// TIA Portal V20 export
FUNCTION "LER_PartData_QrReaderPos" : Void   // FC10000, LAD
// stored: Access Published, SetENOAutomatically false
   VAR_INPUT
      generateCondition : Bool;
      PartOn : Bool;
      JudgmentOK : Bool;
      JudgmentNG : Bool;
      JudgmentBusy : Bool;
      QrReadData : String;
   END_VAR
   VAR_OUTPUT
      PartData : "LER_typePartData";
      ResultData : "LER_typeQrData";
   END_VAR
   VAR_TEMP
      tempRET_VAL : Word;
   END_VAR
   VAR CONSTANT
      PartStatus_Busy : Byte := 16#2;
      PartStatus_Ok : Byte := 16#3;
      PartStatus_NG : Byte := 16#4;
      TRUE : Bool := TRUE;
   END_VAR
   VAR_TEMP   // added for the SCL form of the ladder/FBD networks
      _w1 : Bool;
   END_VAR
BEGIN

REGION Network 1: PartStatus
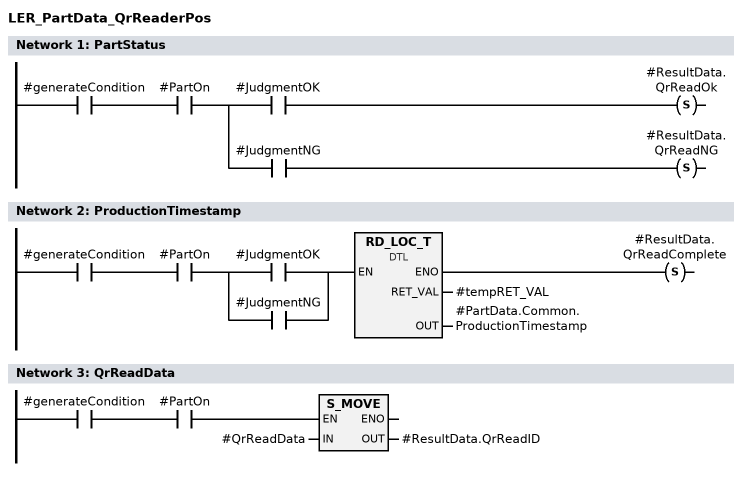
   RUNG wire#powerrail
      Contact( #generateCondition )
      Contact( #PartOn )
      wire#w1
      Contact( #JudgmentOK )
      S_Coil( #ResultData.QrReadOk )
   END_RUNG
   RUNG wire#w1
      Contact( #JudgmentNG )
      S_Coil( #ResultData.QrReadNG )
   END_RUNG
   // the same network as SCL:
   #_w1 := #generateCondition AND #PartOn;
   IF #_w1 AND #JudgmentOK THEN #ResultData.QrReadOk := TRUE; END_IF;
   IF #_w1 AND #JudgmentNG THEN #ResultData.QrReadNG := TRUE; END_IF;
END_REGION

REGION Network 2: ProductionTimestamp
   RUNG wire#powerrail
      Contact( #generateCondition )
      Contact( #PartOn )
      wire#w1
      Contact( #JudgmentOK )
      wire#w2
      { S7_Templates := "date_type := DTL" } RD_LOC_T(RET_VAL => #tempRET_VAL, OUT => #PartData.Common.ProductionTimestamp)
      S_Coil( #ResultData.QrReadComplete )
   END_RUNG
   RUNG wire#w1
      Contact( #JudgmentNG )
   END_RUNG wire#w2
   // the same network as SCL:
   #tempRET_VAL := RD_LOC_T(EN := #generateCondition AND #PartOn AND (#JudgmentOK OR #JudgmentNG),
                           OUT => #PartData.Common.ProductionTimestamp,
                           ENO => #_w1);
   IF #_w1 THEN #ResultData.QrReadComplete := TRUE; END_IF;
END_REGION

REGION Network 3: QrReadData
   RUNG wire#powerrail
      Contact( #generateCondition )
      Contact( #PartOn )
      S_Move(in := #QrReadData, out => #ResultData.QrReadID)
   END_RUNG
   // the same network as SCL:
   IF #generateCondition AND #PartOn THEN #ResultData.QrReadID := #QrReadData; END_IF;
END_REGION
END_FUNCTION
